FUNCTION "LGF_SmoothByPolynomFC" : Void
TITLE = LGF_SmoothByPolynomFC
{ S7_Optimized_Access := 'TRUE' }
AUTHOR : Siemens_Digital_Industry
FAMILY : LGF
NAME : LGF_SmoothByPolynomFC
//This function calculates the smoothed values by polynomial acyclically.
//
//For smoothing, a 3rd degree polynomial is placed through five value points. The error squares of the distances between polynomial and real value are minimized. The smoothed values can be determined from the polynomial parameters obtained in this way.
//
//The function reads an array that is smoothed. $N-4$ smoothed measured values can be calculated from N measured values. The output array contains the value 0 in the index (0,1,N-1,N). However, replacement values can be calculated.
   VAR_OUTPUT
      error : Bool;   // FALSE: No error  TRUE: An error occurred during the execution of the FB
      status : Word;   // 16#0000-16#7FFF: Status of the FB  16#8000-16#FFFF: Error identification (see following Table)
   END_VAR

   VAR_IN_OUT
      values : Array[*] of LReal;   // Values that are to be included in the smoothing.
      smoothedValues : Array[*] of LReal;   // The smoothed values.
   END_VAR

   VAR_TEMP
      tempCount : Int;   // Temp count
      tempNumberOfElements : Int;   // Temp number of elements
      tempNumberOfElementsOut : Int;   // Temp number of elements out
      tempLowerBound : Int;   // Temp lower bound
      tempUpperBound : Int;   // Temp upper bound
      tempLowerBoundOut : Int;   // Temp lower bound out
      tempUpperBoundOut : Int;   // Temp upper bound out
   END_VAR

   VAR CONSTANT
      NUMBER_OF_ELEMENTS_CORRECTION : Int := 1;   // Count also the starting value. e.g. [0.. 9] = 10 elements
      DIMENSION_ONE : UDInt := 1;   // First dimension of the array
      MINIMUM_ARRAY_ELEMENTS : UDInt := 5;   // The needed minimum number of ARRAY elements. Starting from 0
      STATUS_FINISHED_NO_ERROR : Word := 16#0000;   // Status: Execution finished without errors
      ERR_ARRAYS_DIFFERENT : Word := 16#8400;   // Error: The Array sizes are not equal.  The arrays `values` and `smoothedValues` must have the same size.
      ERR_NOT_ENOUGH_VALUES : Word := 16#8401;   // Error: Not enough values.  The block requires five (5) values to calculate a smoothed value. Increase the size of the array at the input parameter `values`. Adapt the array on the output parameter `smoothedValues` to the new size.
   END_VAR


BEGIN
	REGION Block info header
	  //============================================================================
	  // SIEMENS AG / (c)Copyright 2017
	  //----------------------------------------------------------------------------
	  // Title:            LGF_SmoothByPolynomFC
	  // Comment/Function: This function calculates the smoothed values by polynom
	  // Library/Family:   LGF(Library General Functions)
	  // Author:           Siemens Digital Industry Support
	  // Tested with:      S7-PLCSIM Advanced V2.0 SP1
	  // Engineering:      TIA Portal V15 Update 2
	  // Restrictions:     ENO disabled - error handling done by error and status
	  // Requirements:     PLC (S7-1200 / S7-1500)
	  //-------------------------------------------------------------------------------
	  // Change log table:
	  // Version  | Date       | Expert in charge       | Changes applied
	  //----------|------------|------------------------|------------------------------
	  // 01.00.00 | 23.11.2018 | Siemens Industry Online Support
	  //                       | First released version
	  // 01.00.05 | 15.11.2019 | Simatic Systems Support
	  //                       | Regions, comments and constants are added
	  // 03.00.00 | 23.04.2020 | Simatic Systems Support
	  //                       | Set version to V3.0.0, harmonize the version of the whole library
	  // 03.00.01 | 06.04.2021 | Simatic Systems Support
	  //                       | Insert documentation
	  //=============================================================================
	END_REGION Block info header

	REGION DESCRIPTION
	  (/*
	The 3rd degree compensation polynomial is calculated as follows:

	$$
	  \overline{y(n)} = \frac{1}{35} \cdot (-3 \cdot y(n-2) +12 \cdot y(n-1) +17 \cdot y(n) +12 \cdot y(n+1) -3 \cdot y(n+2))
	$$

	$N-4$ smoothed measured values can thus be calculated from the N measured values. The output array contains the value 0 in the index (0.1, N-1, N).

	These “missing” values are calculated with the following formalisms:

	$$
	  \overline{y(n-2)} = \frac{1}{70} \cdot (69 \cdot y(n-2) +4 \cdot y(n-1) -6 \cdot y(n) +4 \cdot y(n+1) -y(n+2))
	$$

	$$
	  \overline{y(n-1)} = \frac{2}{70} \cdot (2 \cdot y(n-2) +27 \cdot y(n-1) +12 \cdot y(n) -8 \cdot y(n+1) +2 \cdot y(n+2))
	$$

	$$
	  \overline{y(n+1)} = \frac{2}{70} \cdot (2 \cdot y(n-2) -8 \cdot y(n-1) +12 \cdot y(n) +27 \cdot y(n+1) +2 \cdot y(n+2))
	$$

	$$
	  \overline{y(n+2)} = \frac{1}{70} \cdot (-y(n-2) +4 \cdot y(n-1) -6 \cdot y(n) +4 \cdot y(n+1) +69 \cdot y(n+2))
	$$
	*/)
	END_REGION DESCRIPTION

	REGION Checking number of lower and upper bound
	  #tempLowerBound := DINT_TO_INT(LOWER_BOUND(ARR := #values, DIM := #DIMENSION_ONE));
	  #tempUpperBound := DINT_TO_INT(UPPER_BOUND(ARR := #values, DIM := #DIMENSION_ONE));

	  #tempNumberOfElements := #tempUpperBound - #tempLowerBound + #NUMBER_OF_ELEMENTS_CORRECTION;

	  #tempLowerBoundOut := DINT_TO_INT(LOWER_BOUND(ARR := #smoothedValues, DIM := #DIMENSION_ONE));
	  #tempUpperBoundOut := DINT_TO_INT(UPPER_BOUND(ARR := #smoothedValues, DIM := #DIMENSION_ONE));

	  #tempNumberOfElementsOut := #tempUpperBoundOut - #tempLowerBoundOut + #NUMBER_OF_ELEMENTS_CORRECTION;

	  //check if size of arrays is ok
	  IF #tempNumberOfElementsOut <> #tempNumberOfElements THEN
	    #error := true;
	    #status := #ERR_ARRAYS_DIFFERENT;
	    RETURN;
	  ELSIF #tempNumberOfElements <= #MINIMUM_ARRAY_ELEMENTS THEN
	    #error := true;
	    #status := #ERR_NOT_ENOUGH_VALUES;
	    RETURN;
	  END_IF;

	  FOR #tempCount := #tempLowerBound + 2 TO #tempUpperBound - 2 DO
	    // calculate new smoothed value
	    // keep the "Magic Numbers" as they are part of the Math equation and would extent the formular in a unreadable way
	    // y(n)=1/35*(-3*y(n-2)+12*y(n-1)+17*y(n)+12*y(n+1)-3*y(n+2))
	    // 1/35 = 0.028571
	    #smoothedValues[#tempCount] := 0.028571 * (-3 * #values[#tempCount - 2] + 12 * #values[#tempCount - 1] + 17 * #values[#tempCount] + 12 * #values[#tempCount + 1] - 3 * #values[#tempCount + 2]);
	  END_FOR;

	  // calculate Replacementvalues for 0,1 and n-1,n
	  // y(0) =1/70*(69*y(0)+4*y(1)-6*y(2)+4*y(3)-y(4))
	  // 1/70 = 0.014286
	  #smoothedValues[#tempLowerBound] := 0.014286 * (69 * #values[#tempLowerBound] + 4 * #values[#tempLowerBound + 1] - 6 * #values[#tempLowerBound + 2] + 4 * #values[#tempLowerBound + 3] - #values[#tempLowerBound + 4]);
	  // y(1) =2/70*(2*y(0)+27*y(1)+12*y(2)-8*y(3)+2*y(4))
	  // 2/70 = 0.028571
	  #smoothedValues[#tempLowerBound + 1] := 0.028571 * (2 * #values[#tempLowerBound] + 27 * #values[#tempLowerBound + 1] + 12 * #values[#tempLowerBound + 2] - 8 * #values[#tempLowerBound + 3] + 2 * #values[#tempLowerBound + 4]);
	  // y(n-1) =2/70*(2*y(n-4)-8*y(n-3)+12*y(n-2)+27*y(n-1)+2*y(n))
	  // 2/70 = 0.028571
	  #smoothedValues[#tempUpperBound - 1] := 0.028571 * (2 * #values[#tempUpperBound - 4] - 8 * #values[#tempUpperBound - 3] + 12 * #values[#tempUpperBound - 2] + 27 * #values[#tempUpperBound - 1] + 2 * #values[#tempUpperBound]);
	  // y(n) =1/70*(-y(n-4)+4*y(n-3)-6*y(n-2)+4*y(n-1)+69*y(n))
	  // 1/70 = 0.014286
	  #smoothedValues[#tempUpperBound] := 0.014286 * (- #values[#tempUpperBound - 4] + 4 * #values[#tempUpperBound - 3] - 6 * #values[#tempUpperBound - 2] + 4 * #values[#tempUpperBound - 1] + 69 * #values[#tempUpperBound]);

	  #error := false;
	  #status := #STATUS_FINISHED_NO_ERROR;
	  // ENO mechanism is not used - forced to true.
	  ENO := TRUE;
	END_REGION

END_FUNCTION

